// TwinCAT 3 PLC project FileIO
// ProgramVersion: 3.1.4020.10
// libraries:
//   Tc2_Standard, * (Beckhoff Automation GmbH)
//   Tc2_System, * (Beckhoff Automation GmbH)
//   Tc3_Interfaces, * (Beckhoff Automation GmbH)
//   Tc3_Module, * (Beckhoff Automation GmbH)
// project tree:
//   FileIO/ FunctionResult_Log.TcDUT, MachineLog.TcPOU
// (motion and I/O tree: see PLC project motion_library)
// real-time tasks:
//   TASK PlcTask: cycle T#10ms, priority 20, ADS port 350

// ---- FileIO/FunctionResult_Log.TcDUT
TYPE FunctionResult_Log :
(
	ERROR := -1,
	BUSY := 0,
	DONE
);
END_TYPE

// ---- FileIO/MachineLog.TcPOU
FUNCTION_BLOCK MachineLog
VAR
	fbOpenFile: FB_FileOpen;
	fbCloseFile: FB_FileClose;
	fbPutInFile: FB_FilePuts;
	hFileHandle: UINT;
	fbGetTime: NT_GetTime;
	CurrentTime: TIMESTRUCT;
	CurrentTime_String: STRING(24);
	WriteState: INT := 0;
	LogDelimiter: STRING(5) := ',';
	LogEOL: STRING(5) := '$R$N';
END_VAR

;

{attribute 'object_name' := 'CloseFile'}
METHOD CloseFile : FunctionResult_Log
fbCloseFile(
	sNetId:= '', 
	hFile:= hFileHandle, 
	bExecute:= TRUE, 
	tTimeout:= T#1S );
	
IF fbCloseFile.bError THEN
	fbCloseFile( 
		bExecute:= FALSE );
	WriteState := -1;
CloseFile := FunctionResult_Log.ERROR;
END_IF

IF NOT fbCloseFile.bBusy AND NOT fbCloseFile.bError THEN
	fbCloseFile( 
		bExecute:= FALSE );
	hFileHandle := 0;
	WriteState := WriteState + 1;
	CloseFile := FunctionResult_Log.DONE;
END_IF

CloseFile := FunctionResult_Log.BUSY;
END_METHOD

{attribute 'object_name' := 'CreateEntry'}
METHOD CreateEntry : FunctionResult_Log
VAR_INPUT
	EntryMessage: STRING(255);
END_VAR
VAR
	Buffer: STRING(500);
END_VAR
CASE WriteState OF 
	-1	:	CreateEntry := FunctionResult_Log.BUSY;
	0	:	OpenFile('C:\Users\SiangC\Desktop\Test.txt');
	1	:	GetTime();
	2	:	WriteToFile(EntryMessage);
	3	:	CloseFile();
	4	:	IF Reset() = FunctionResult_Log.DONE THEN CreateEntry := FunctionResult_Log.DONE; END_IF
END_CASE
END_METHOD

PROPERTY Delimiter : STRING(5)
GET
Delimiter := LogDelimiter;
END_GET
SET
LogDelimiter := Delimiter;
END_SET
END_PROPERTY

{attribute 'object_name' := 'EntryBuilder'}
METHOD PRIVATE EntryBuilder : STRING(255)
VAR_INPUT
	MESSAGE_COMPONENT: ARRAY[0..3] OF STRING(255);
END_VAR
VAR
	BUFFER: STRING(255);
	i: INT;
END_VAR
BUFFER := CONCAT(MESSAGE_COMPONENT[0],MESSAGE_COMPONENT[1]);
FOR i := 2 TO 3 BY 1 DO
	BUFFER := CONCAT(BUFFER,MESSAGE_COMPONENT[i]);
END_FOR
EntryBuilder := BUFFER;
END_METHOD

PROPERTY EOL : STRING(5)
GET
EOL := LogEOL;
END_GET
SET
LogEOL := EOL;
END_SET
END_PROPERTY

{attribute 'object_name' := 'GetTime'}
METHOD PRIVATE GetTime : FunctionResult_Log
(*
	Get the system's time
		-> Output to CurrentTime (TIMESTRUCT)
*)
fbGetTime(
			NETID:= '', 
			START:= TRUE, 
			TMOUT:= T#1S, 
			TIMESTR=> CurrentTime);
(*
	If error occurs
		-> Reset the Execute input
		-> Advance object state to its error state (-1)
*)
IF fbGetTIme.ERR THEN
	fbGetTime( 
		START:= FALSE );
	WriteState := -1;
	GetTime := FunctionResult_Log.ERROR;
END_IF

(*
	If successful
		-> Reset the Execute input
		-> Convert time to STRING(24) format 
		-> Advance object state (++)
*)
IF NOT fbGetTime.BUSY AND NOT fbGetTime.ERR THEN
	fbGetTime( 
		START:= FALSE );
	CurrentTime_String := SYSTEMTIME_TO_STRING(CurrentTime);
	WriteState := WriteState + 1;
	GetTime := FunctionResult_Log.DONE;
END_IF

(*
	Returns busy otherwise
*)
GetTime := FunctionResult_Log.BUSY;
END_METHOD

{attribute 'object_name' := 'OpenFile'}
METHOD PRIVATE OpenFile : FunctionResult_Log
VAR_INPUT
	sFilePath: T_MAXSTRING;
END_VAR
(*
	Executes the function block.
		-> Obtain the File Handle and store it in hFileHandle (UINT)
		-> File Handle is used by other File IO function blocks
*)
fbOpenFile(
	sNetId:= '', 
	sPathName:= sFilePath, 
	nMode:= FOPEN_MODEAPPEND OR FOPEN_MODEPLUS, 
	ePath:= PATH_GENERIC, 
	bExecute:= TRUE, 
	tTimeout:= T#1S,  
	hFile=> hFileHandle);
	
(*
	If error occurs.
		-> Reset the Execute input.
		-> Advance the object state to its Error state (-1)
*)
IF fbOpenFile.bError THEN 
	fbOpenFile(
		bExecute:= FALSE );
	WriteState := -1;
	OpenFile := FunctionResult_Log.ERROR;
END_IF

(*
	Function block is complete if it is 
		a) NOT BUSY
		b) NO ERROR
		-> Reset the Execute input
		-> Advance the object state to the next state (++)
*)
IF NOT fbOpenFile.bBusy AND NOT fbOpenFile.bError AND hFileHandle > 0 THEN
	fbOpenFile(
		bExecute:= FALSE );
	WriteState := WriteState + 1;
	OpenFile := FunctionResult_Log.DONE;
END_IF

(*
	Otherwise returns Busy signal
*)
OpenFile := FunctionResult_Log.BUSY;
END_METHOD

{attribute 'object_name' := 'Reset'}
METHOD Reset : FunctionResult_Log
fbCloseFile( 
	bExecute:= FALSE );
fbOpenFile(
	bExecute:= FALSE );
fbPutInFile(
	bExecute:= FALSE );
WriteState := 0;
Reset := FunctionResult_Log.DONE;
END_METHOD

{attribute 'object_name' := 'WriteToFile'}
METHOD PRIVATE WriteToFile : FunctionResult_Log
VAR_INPUT
	MESSAGE: STRING(255);
END_VAR
VAR
	MESSAGE_BUFFER: ARRAY[0..3] OF STRING(255) := [CurrentTime_String, Delimiter, MESSAGE, LogEOL];
	BUFFER: T_MAXSTRING;
END_VAR
fbPutInFile(
	sNetId:= '', 
	hFile:= hFileHandle, 
	sLine:= EntryBuilder(MESSAGE_BUFFER), 
	bExecute:= TRUE, 
	tTimeout:= T#1S );
	
IF fbPutInFile.bError THEN
	fbPutInFile(
		bExecute:= FALSE );
	WriteState := -1;
	WriteToFile := FunctionResult_Log.ERROR;
END_IF	

IF NOT fbPutInFile.bBusy AND NOT fbPutInFile.bError THEN
	fbPutInFile(
		bExecute:= FALSE );
	WriteState := WriteState + 1;
	WriteToFile := FunctionResult_Log.DONE;
END_IF

WriteToFile := FunctionResult_Log.BUSY;
END_METHOD

END_FUNCTION_BLOCK
